TYPE DB_FunctionResult :
(
	DB_Ok := -1,
	DB_Error,
	DB_Busy
);
END_TYPE

(* stored: Version 1.1.0.1, ProductVersion 3.1.0.36
   DUT DB_FunctionResult: Id {42a0b938-4162-41c0-8e0c-6b57f8215596} *)
